TYPE ST_BalluffDevice :
STRUCT
	ErrorRegister	: BYTE;
	Temperature	: INT;
	
END_STRUCT
END_TYPE

(* stored: Version 1.1.0.1, ProductVersion 3.1.4020.12
   DUT ST_BalluffDevice: Id {bf27cdb9-fa26-410b-8013-0b2e3be721d2} *)
